(* IEC 61131-3 sources: std_i2980_v2.06_cp053/Source/IMM/ieccontrol/InjectionGeneral (part 10) *)

bUsePosDetect := TRUE;

@SaText @RT(19)AInitDecompInterPos 1 @TL(24)
(**************************************** WARNING ********************************************
 *** The KEBA Kemro K2 System including software is not intended for safety control tasks! ***
 ***                       For further information see Comment tab!                        ***
 *********************************************************************************************)

abDecompInterPos.aRun(bStart := FALSE);
abDecompSetupServo.aRun(bStart := FALSE);

IF sv_DecompInterPosSettings.Mode = nTimeDependent THEN
   //set target position to maximum value
   //-> screw ramps down to maximum position no matter if the
   //move time is set to a high value
   rTargetPosition := sv_rScrewStroke;

   //set movement time
   abDecompInterPos.aSetMoveTime(dSetMoveTime := sv_DecompInterPosSettings.dDecompTime);
ELSE
   //mode position dependent -> set according target value
   aVolumeToDistance(rVolume := sv_DecompInterPosSettings.rDecompPos,
                     rDistance => rTargetPosition);
END_IF;

bUsePosDetect := TRUE;

@SaText @RT(16)AResetIdentBlock 1 @TL(12)
abDecompStep.aRun(bStart := FALSE);

rTargetPosition := sv_rIdentPosition;
bUsePosDetect := (sv_rIdentPosition <> 0.0);

abDecompSetupServo.aRun(bStart := FALSE);
IF  abDecompStep.aRun.bError OR abDecompSetupServo.aRun.bError THEN
   sv_CalibState.Status := tnCalibState_Error;
   bError := TRUE;
   dummy := Print("Ident Error: Reset calib block failed");
END_IF;

@SaText @RT(22)ADecompSetupServoIdent 1 @TL(14)
IF sv_IMM_Type = nKAPPL_IMM_ServoValve THEN
   abDecompSetupServo.aRun(bStart := TRUE,
                           bStop := bStop,
                           bDirection := TRUE,
                           rActPos := sv_rScrewPositionAbs,
                           rTargetPos := rTargetPosition,
                           bUsePosDetect := bUsePosDetect,
                           rStartOutputPre := 0.0,
                           rStartOutputVel := 0.0,
                           dDelayTimeOn := T#0s,
                           dDelayTimeOff := T#0s);
   sv_rServoOutput := abDecompSetupServo.aRun.rOutputVel;
END_IF;

@SaText @RT(16)ATransducerCalib 1 @TL(30)
(**************************************** WARNING ********************************************
 *** The KEBA Kemro K2 System including software is not intended for safety control tasks! ***
 ***                       For further information see Comment tab!                        ***
 *********************************************************************************************)

// Calibration works with stroke not volume
abScrewBwdCalib.aRun(bStop := bStop OR sv_bTransducerError,
                     bStart := TRUE,
                     rActVoltage := ai_Position,
                     rMaxVoltageDiff := sv_rMaxVoltageDiff,
                     dStandStillDetectTime := sv_dStandStillDetectTime,
                     LintabPoint := sv_TmpLintabPoint,
                     rSetValue := sv_rScrewStroke,
                     dDelayTimeOn := sv_DecompTimesSet.dSetDelayTimePump,
                     dDelayTimeOff := sv_DecompTimesSet.dSetDelayTimeValve,
                     bActive => sv_bOutputActive,
                     rOutputPre => rPressureAbs,
                     rOutputVel => rVelocityAbs,
                     bPreOutputReached => sv_bPreOutputReady,
                     iErrorInfo => iErrorInfo);

sv_bDoTransducerCalib := NOT (abScrewBwdCalib.aRun.bPointDetected);
bError := abScrewBwdCalib.aRun.bError OR bError;

abLintabApplyPres.aCalc(rX := rPressureAbs,
                        rY => sv_rPressure);

abLintabApplyVel.aCalc(rX := rVelocityAbs,
                       rY => sv_rVelocity);

@SaText @RT(11)AStepOutput 1 @TL(32)
(**************************************** WARNING ********************************************
 *** The KEBA Kemro K2 System including software is not intended for safety control tasks! ***
 ***                       For further information see Comment tab!                        ***
 *********************************************************************************************)

abDecompStep.aRun(bUsePosDetect := (sv_rIdentPosition <> 0.0),
                  rPositionDown := (sv_rScrewPositionAbs + sv_rIdentPosition) * 0.5,
                  rLowOutput := sv_rMaxSpeedBwd * 0.1,
                  bStart := TRUE,
                  bStop := bStop,
                  bDirection := TRUE,
                  rActPos := sv_rScrewPositionAbs,
                  rTargetPos := sv_rIdentPosition,
                  dDelayTimeOn := sv_DecompTimesSet.dSetDelayTimePump,
                  dDelayTimeOff := sv_dSetDelayTimeOffBwd,
                  rPositionUp := sv_rScrewPositionAbs,
                  rHighOutput := sv_ConstDecompSetup.Velocity.Output.rOutputValue,
                  dMaxMoveTime := sv_DecompTimesSet.dMaxMoveTime,
                  rStopRamp := sv_rIdentStopRamp,
                  bActive => sv_bOutputActive,
                  rOutputPre => rPressureAbs,
                  rOutputVel => rVelocityAbs,
                  bPreOutputReached => sv_bPreOutputReady);

sv_rVelocityAbs := rVelocityAbs;

abLintabApplyPres.aCalc(rX := rPressureAbs,
                        rY => sv_rPressure);

abLintabApplyVel.aCalc(rX := rVelocityAbs,
                       rY => sv_rVelocity);

@SaText @RT(12)ADecompSetup 1 @TL(26)
(**************************************** WARNING ********************************************
 *** The KEBA Kemro K2 System including software is not intended for safety control tasks! ***
 ***                       For further information see Comment tab!                        ***
 *********************************************************************************************)

abDecompSetup.aRun(bStart := TRUE,
                   bStop := bStop,
                   bDirection := TRUE,
                   rActPos := sv_rScrewPositionAbs,
                   rTargetPos := rTargetPosition,
                   bUsePosDetect := bUsePosDetect,
                   dMaxTime := dMaxMoveTime,
                   dDelayTimeOn := sv_DecompTimesSet.dSetDelayTimePump,
                   dDelayTimeOff := sv_DecompTimesSet.dSetDelayTimeValve,
                   rOutputPre => rPressureAbs,
                   rOutputVel => rVelocityAbs,
                   bActive => sv_bOutputActive,
                   bPreOutputReached => sv_bPreOutputReady);

abLintabApplyPres.aCalc(rX := rPressureAbs);
b := WRITE_SVREAL_DIRECT(sv_rPressure, abLintabApplyPres.aCalc.rY);

abLintabApplyVel.aCalc(rX := rVelocityAbs);
b := WRITE_SVREAL_DIRECT(sv_rVelocity, abLintabApplyVel.aCalc.rY);

@SaText @RT(12)ADecompPurge 1 @TL(25)
(**************************************** WARNING ********************************************
 *** The KEBA Kemro K2 System including software is not intended for safety control tasks! ***
 ***                       For further information see Comment tab!                        ***
 *********************************************************************************************)

abDecompPurge.aRun(bStart := TRUE,
                   bStop := bStop,
                   bDirection := TRUE,
                   rActPos := sv_rScrewPositionAbs,
                   rTargetPos := rTargetPosition,
                   bUsePosDetect := TRUE,
                   dDelayTimeOn := sv_DecompTimesSet.dSetDelayTimePump,
                   dDelayTimeOff := sv_DecompTimesSet.dSetDelayTimeValve,
                   rOutputPre => rPressureAbs,
                   rOutputVel => rVelocityAbs,
                   bActive => sv_bOutputActive,
                   bPreOutputReached => sv_bPreOutputReady);

abLintabApplyPres.aCalc(rX := rPressureAbs);
b := WRITE_SVREAL_DIRECT(sv_rPressure, abLintabApplyPres.aCalc.rY);

abLintabApplyVel.aCalc(rX := rVelocityAbs);
b := WRITE_SVREAL_DIRECT(sv_rVelocity, abLintabApplyVel.aCalc.rY);

@SaText @RT(15)ADecompInterPos 1 @TL(29)
(**************************************** WARNING ********************************************
 *** The KEBA Kemro K2 System including software is not intended for safety control tasks! ***
 ***                       For further information see Comment tab!                        ***
 *********************************************************************************************)

abDecompInterPos.aRun(bStop := bStop OR sv_bTransducerError OR (sv_DecompInterPosSettings.Mode = nNotUsed),
                      bStart := TRUE,
                      bDirection := TRUE,
                      rActPos := sv_rScrewPositionAbs,
                      rTargetPos := rTargetPosition,
                      bUsePosDetect := TRUE,
                      dMaxTime := sv_DecompTimesSet.dMaxMoveTime,
                      dDelayTimeOn := sv_DecompTimesSet.dSetDelayTimePump,
                      dDelayTimeOff := sv_DecompTimesSet.dSetDelayTimeValve,
                      rOutputPre => rPressureAbs,
                      rOutputVel => rVelocityAbs,
                      bActive => sv_bOutputActive,
                      bPreOutputReached => sv_bPreOutputReady);

b := WRITE_SV_DIRECT(sv_DecompTimesAct.dActMoveTime, abDecompInterPos.aRun.dActTime);
b := WRITE_SV_DIRECT(sv_ActiveTimesDecompInterPos[g_MoveCtrl.iCount], sv_DecompTimesAct.dActMoveTime);

abLintabApplyPres.aCalc(rX := rPressureAbs);
b := WRITE_SVREAL_DIRECT(sv_rPressure, abLintabApplyPres.aCalc.rY);

abLintabApplyVel.aCalc(rX := rVelocityAbs);
b := WRITE_SVREAL_DIRECT(sv_rVelocity, abLintabApplyVel.aCalc.rY);

@SaText @RT(15)ADecompBefPlast 1 @TL(28)
(**************************************** WARNING ********************************************
 *** The KEBA Kemro K2 System including software is not intended for safety control tasks! ***
 ***                       For further information see Comment tab!                        ***
 *********************************************************************************************)

abDecompBefPlast.aRun(bStop := bStop OR sv_bTransducerError OR (sv_DecompBefPlastSettings.Mode = nNotUsed),
                      bStart := TRUE,
                      bDirection := TRUE,
                      rActPos := sv_rScrewPositionAbs,
                      rTargetPos := rTargetPosition,
                      bUsePosDetect := TRUE,
                      dMaxTime := sv_DecompTimesSet.dMaxMoveTime,
                      dDelayTimeOn := sv_DecompTimesSet.dSetDelayTimePump,
                      dDelayTimeOff := sv_DecompTimesSet.dSetDelayTimeValve,
                      rOutputPre => rPressureAbs,
                      rOutputVel => rVelocityAbs,
                      bActive => sv_bOutputActive,
                      bPreOutputReached => sv_bPreOutputReady);

b := WRITE_SV_DIRECT(sv_dActDecompBeforeTime, abDecompBefPlast.aRun.dActTime);
b := WRITE_SV_DIRECT(sv_DecompTimesAct.dActMoveTime, sv_dActDecompBeforeTime);

abLintabApplyPres.aCalc(rX := rPressureAbs);
b := WRITE_SVREAL_DIRECT(sv_rPressure, abLintabApplyPres.aCalc.rY);

abLintabApplyVel.aCalc(rX := rVelocityAbs);
b := WRITE_SVREAL_DIRECT(sv_rVelocity, abLintabApplyVel.aCalc.rY);

@SaText @RT(15)ADecompAftPlast 1 @TL(29)
(**************************************** WARNING ********************************************
 *** The KEBA Kemro K2 System including software is not intended for safety control tasks! ***
 ***                       For further information see Comment tab!                        ***
 *********************************************************************************************)

abDecompAftPlast.aRun(bStop := bStop OR sv_bTransducerError OR (sv_DecompAftPlastSettings.Mode = nNotUsed),
                      bStart := TRUE,
                      bDirection := TRUE,
                      rActPos := sv_rScrewPositionAbs,
                      rTargetPos := rTargetPosition,
                      bUsePosDetect := TRUE,
                      dMaxTime := sv_DecompTimesSet.dMaxMoveTime,
                      dDelayTimeOn := sv_DecompTimesSet.dSetDelayTimePump,
                      dDelayTimeOff := sv_DecompTimesSet.dSetDelayTimeValve,
                      rOutputPre => rPressureAbs,
                      rOutputVel => rVelocityAbs,
                      bActive => sv_bOutputActive,
                      bPreOutputReached => sv_bPreOutputReady);

b := WRITE_SV_DIRECT(sv_dActDecompAfterTime, abDecompAftPlast.aRun.dActTime);
b := WRITE_SV_DIRECT(sv_DecompTimesAct.dActMoveTime, sv_dActDecompAfterTime);

abLintabApplyPres.aCalc(rX := rPressureAbs);
b := WRITE_SVREAL_DIRECT(sv_rPressure, abLintabApplyPres.aCalc.rY);

abLintabApplyVel.aCalc(rX := rVelocityAbs);
b := WRITE_SVREAL_DIRECT(sv_rVelocity, abLintabApplyVel.aCalc.rY);

@SaTrans 0
@SaExits 0
@END_SfcBody

@@@BEG_Comment@@@
@TL(4)
This algorithm is responsible for executing the movement.
Depending on MoveId, OperationMode and activated transducer calibration the according
movement is executed.
The different actions contain the movement blocks and the according parameters.
@@@END_Comment@@@

@BEG_Body
@TL(50)
(**************************************** WARNING ********************************************
 *** The KEBA Kemro K2 System including software is not intended for safety control tasks! ***
 ***                       For further information see Comment tab!                        ***
 *********************************************************************************************)

// Decomp. after plast:
abDecompAftPlast.aInit(pConst := @sv_DecompAftPlastSettings.ConstOutput,
                       MoveId := cMoveDecompAftPlast,
                       pdCalcedDuration := @sv_dCalculatedDurationDecompAft,
                       prCalcDurationStartPosition := @sv_rDecompAftCalcDurStartPos,
                       prCalcDurationEndPosition := @sv_rDecompAftCalcDurEndPos);

// Decomp before plast:
abDecompBefPlast.aInit(pConst := @sv_DecompBefPlastSettings.ConstOutput,
                       MoveId := cMoveDecompBefPlast,
                       pdCalcedDuration := @sv_dCalculatedDurationDecompBef,
                       prCalcDurationStartPosition := @sv_rDecompBefCalcDurStartPos,
                       prCalcDurationEndPosition := @sv_rDecompBefCalcDurEndPos);

// Decomp setup:
abDecompSetup.aInit(pConst := @sv_ConstDecompSetup,
                    MoveId := cMoveDecompAftPlast);

// Decomp setup servo:
abDecompSetupServo.aInit(pConst := @sv_ConstDecompSetupServo,
                         MoveId := cMoveDecompAftPlast);

// Decomp interpos:
abDecompInterPos.aInit(pConst := @sv_DecompInterPosSettings.ConstOutput,
                       MoveId := cMoveDecompInterPos);

// Init bwd calib:
abScrewBwdCalib.aInit(pConst := @sv_ConstDecompSetup,
                      MoveId := cMoveDecompAftPlast);

// Init decomp for purge:
abDecompPurge.aInit(pConst := @sv_PurgeSettings.DecompParams.ConstOutput,
                    MoveId := cMoveDecompPurge);

// Init lintab apply press:
abLintabApplyPres.aInit(pLintab := @sv_LintabOutBwdP);

// Init lintab apply vel
abLintabApplyVel.aInit(pLintab := @sv_LintabOutBwdV);

// Init ident. movement:
abDecompStep.aInit(pConst := @sv_ConstDecompSetup,
                   MoveId := cMoveDecompAftPlast,
                   prMaxSpeed := @sv_rMaxSpeedBwd);

@END_Body

@@@BEG_Comment@@@
@TL(0)

@@@END_Comment@@@

@BEG_Body
@TL(10)
(**************************************** WARNING ********************************************
 *** The KEBA Kemro K2 System including software is not intended for safety control tasks! ***
 ***                       For further information see Comment tab!                        ***
 *********************************************************************************************)

rSize := FCalcScrewSize(sv_rScrewDiameter);
rTime := LINT_TO_REAL(TIME_TO_LINT(dTime)) / 1000000.0;

rVolume := (rVelocity * rTime * rSize) / 1000.0;

@END_Body

@@@BEG_Comment@@@
@TL(2)
calculate an estimated volume considering constant velocity over a defined time
ramps are not considered in this calculation
@@@END_Comment@@@

@BEG_Body
@TL(17)
(**************************************** WARNING ********************************************
 *** The KEBA Kemro K2 System including software is not intended for safety control tasks! ***
 ***                       For further information see Comment tab!                        ***
 *********************************************************************************************)

//copy minoutput to decomp before plast settings
sv_DecompBefPlastSettings.ConstOutput.Velocity.rMinOutput := sv_MinOutputDecomp.rVelocity;
sv_DecompBefPlastSettings.ConstOutput.Pressure.rMinOutput := sv_MinOutputDecomp.rPressure;

//copy minoutput to decomp after plast settings
sv_DecompAftPlastSettings.ConstOutput.Velocity.rMinOutput := sv_MinOutputDecomp.rVelocity;
sv_DecompAftPlastSettings.ConstOutput.Pressure.rMinOutput := sv_MinOutputDecomp.rPressure;

//copy minoutput to decomp movement in setup mode
sv_ConstDecompSetup.Velocity.rMinOutput := sv_MinOutputDecomp.rVelocity;
sv_ConstDecompSetup.Pressure.rMinOutput := sv_MinOutputDecomp.rPressure;

@END_Body

@@@BEG_Comment@@@
@TL(0)

@@@END_Comment@@@

@BEG_Body
@TL(8)
(**************************************** WARNING ********************************************
 *** The KEBA Kemro K2 System including software is not intended for safety control tasks! ***
 ***                       For further information see Comment tab!                        ***
 *********************************************************************************************)

mrDecAftPlastEnd := sv_PlastProfVis.Profile.Points[(sv_PlastProfVis.Profile.iNoOfPoints+1)].rStartPos +
                    sv_DecompAftPlastSettings.rDecompPos;

@END_Body

@@@BEG_Comment@@@
@TL(0)

@@@END_Comment@@@

@BEG_Body
@TL(13)
(**************************************** WARNING ********************************************
 *** The KEBA Kemro K2 System including software is not intended for safety control tasks! ***
 ***                       For further information see Comment tab!                        ***
 *********************************************************************************************)

// set flags that indicate if movement should be activated
// if false a start movement event is ignored by ABControl

sv_bActivatedDecompBeforePlast := sv_DecompBefPlastSettings.Mode <> nNotUsed;
// Decompression should be possible in SetupMode
sv_bActivatedDecompAfterPlast := (sv_DecompAftPlastSettings.Mode <> nNotUsed) OR
                                 (sv_OperationMode = nSetup);

@END_Body

@@@BEG_Comment@@@
@TL(0)

@@@END_Comment@@@

@BEG_Body
@TL(32)
(**************************************** WARNING ********************************************
 *** The KEBA Kemro K2 System including software is not intended for safety control tasks! ***
 ***                       For further information see Comment tab!                        ***
 *********************************************************************************************)

//plast endposition is maximum value of decomp before and plast profile
rPlastEnd := MAX((sv_PlastProfVis.Profile.Points[sv_PlastProfVis.Profile.iNoOfPoints + 1].rStartPos),
                 sv_rTargetValueDecBefPlast);

IF (sv_DecompAftPlastSettings.Mode = nTimeDependent) THEN
   //calculate estimated target position
   aCalcEstimatedVolume(rVelocity := sv_DecompAftPlastSettings.ConstOutput.Velocity.Output.rOutputValue,
                        dTime := sv_DecompAftPlastSettings.dDecompTime);
   sv_rTargetValueDecAftPlast := MIN((aCalcEstimatedVolume.rVolume + rPlastEnd),sv_rScrewVolume);

ELSIF (sv_DecompAftPlastSettings.Mode = nPosDependent) THEN

   sv_rTargetValueDecAftPlast := sv_DecompAftPlastSettings.rDecompPos + rPlastEnd;

ELSIF sv_DecompAftPlastSettings.Mode = nNotUsed THEN

   sv_rTargetValueDecAftPlast := MAX(rPlastEnd, sv_rTargetValueDecBefPlast);
   b := WRITE_SV_DIRECT(sv_dActDecompAfterTime, dNull);
END_IF;

//convert start position and endposition to mm (startposition = plast endposition)
aVolumeToDistance(rVolume := rPlastEnd);
sv_rDecompAftCalcDurStartPos := aVolumeToDistance.rDistance;

aVolumeToDistance(rVolume := sv_rTargetValueDecAftPlast);
sv_rDecompAftCalcDurEndPos := aVolumeToDistance.rDistance;

@END_Body

@@@BEG_Comment@@@
@TL(0)

@@@END_Comment@@@

@BEG_Body
@TL(29)
(**************************************** WARNING ********************************************
 *** The KEBA Kemro K2 System including software is not intended for safety control tasks! ***
 ***                       For further information see Comment tab!                        ***
 *********************************************************************************************)

IF (sv_DecompBefPlastSettings.Mode = nTimeDependent) THEN

   //calculate estimated target position
   aCalcEstimatedVolume(rVelocity := sv_DecompBefPlastSettings.ConstOutput.Velocity.Output.rOutputValue,
                        dTime := sv_DecompBefPlastSettings.dDecompTime);
   sv_rTargetValueDecBefPlast := MIN(aCalcEstimatedVolume.rVolume,sv_rScrewVolume);

ELSIF (sv_DecompBefPlastSettings.Mode = nPosDependent) THEN

   sv_rTargetValueDecBefPlast := sv_DecompBefPlastSettings.rDecompPos;

ELSIF sv_DecompBefPlastSettings.Mode = nNotUsed THEN

   //decomp not used
   sv_rTargetValueDecBefPlast := 0.0;
   b := WRITE_SV_DIRECT(sv_dActDecompBeforeTime, dNull);
END_IF;

sv_rDecompBefCalcDurStartPos := 0.0;

//convert endposition to mm
aVolumeToDistance(rVolume := sv_rTargetValueDecBefPlast);
sv_rDecompBefCalcDurEndPos := aVolumeToDistance.rDistance;

@END_Body

@@@BEG_Comment@@@
@TL(0)

@@@END_Comment@@@

@BEG_Body
@TL(23)
(**************************************** WARNING ********************************************
 *** The KEBA Kemro K2 System including software is not intended for safety control tasks! ***
 ***                       For further information see Comment tab!                        ***
 *********************************************************************************************)

//avoid out of range errors
i := MAX(1,iInstance);

//copy data of according instance to sv_DecompInterPosSettings
IF sv_InstanceDataDecompInterPos[i].Mode = nDecompTimeDependent THEN
   sv_DecompInterPosSettings.Mode := nTimeDependent;
ELSIF sv_InstanceDataDecompInterPos[i].Mode = nDecompPosDependent THEN
   sv_DecompInterPosSettings.Mode := nPosDependent;
END_IF;

sv_DecompInterPosSettings.dDecompTime := sv_InstanceDataDecompInterPos[i].dTime;
sv_DecompInterPosSettings.rDecompPos := sv_InstanceDataDecompInterPos[i].rTargetValue;
sv_DecompInterPosSettings.ConstOutput.Pressure.Output.rOutputValue := sv_InstanceDataDecompInterPos[i].rPressure;
sv_DecompInterPosSettings.ConstOutput.Velocity.Output.rOutputValue := sv_InstanceDataDecompInterPos[i].rVelocity;

sv_MoveDecompInterPos.pdCalculatedDuration := @sv_InstanceDataDecompInterPos[i].dCalculatedDuration;
sv_MoveDecompInterPos.pdStartDelaySet := @sv_InstanceDataDecompInterPos[i].dDelay;

@END_Body

@@@BEG_Comment@@@
@TL(1)
copy settings of instance to the systemvariable that is used for the movement
@@@END_Comment@@@

@BEG_Body
@TL(10)
(**************************************** WARNING ********************************************
 *** The KEBA Kemro K2 System including software is not intended for safety control tasks! ***
 ***                       For further information see Comment tab!                        ***
 *********************************************************************************************)

IF evStartData.DeviceId = sv_DeviceId AND evStartData.MoveId = cMoveDecompInterPos THEN
   aGetInstanceData(iInstance := evStartData.IntermediateCond);
   miDecompInstance := MAX(1,evStartData.IntermediateCond);
END_IF;

@END_Body

@@@BEG_Comment@@@
@TL(4)
get instance data if start event is received

attention:
taskslot is asigned to make sure that execution is done before evaStart in ABControl.pu
@@@END_Comment@@@

@BEG_Body
@TL(8)
(**************************************** WARNING ********************************************
 *** The KEBA Kemro K2 System including software is not intended for safety control tasks! ***
 ***                       For further information see Comment tab!                        ***
 *********************************************************************************************)

mrDecBefPlastEnd := MIN(sv_rHoldPosition + sv_DecompBefPlastSettings.rDecompPos,
                        sv_PlastProfVis.Profile.Points[(sv_PlastProfVis.Profile.iNoOfPoints+1)].rStartPos);

@END_Body

@@@BEG_Comment@@@
@TL(0)

@@@END_Comment@@@
@END_Body

@END_Contents
